// TIA Portal V16 export
// export: Created 2021-03-05T14:22:14.2551895Z, ExportSetting WithDefaults, DisplayName Totally Integrated Automation Portal, DisplayVersion V16, DisplayName TIA Portal Version Control Interface, DisplayVersion V16, DisplayName TIA Portal Openness, DisplayVersion V16, DisplayName SINAMICS Startdrive Advanced, DisplayVersion V16, DisplayName SINAMICS Startdrive G130, G150, S120, S150, SINAMICS MV, S210, DisplayVersion V16, DisplayName SINAMICS Startdrive G110M, G120, G120C, G120D, G120P, DisplayVersion V16, DisplayName STEP 7 Professional, DisplayVersion V16, DisplayName STEP 7 Safety, DisplayVersion V16, DisplayName WinCC Professional, DisplayVersion V16
TYPE "udtDigitalOutput"
// stored: IsFailsafeCompliant false
   STRUCT
      bAutoVal { ExternalVisible := 'False'; ExternalWritable := 'False'} : Bool;   // Value set by the program
      bOverrideVal { ExternalVisible := 'False'} : Bool;   // Value set by the user, tracks bAuto when bOverrideEnable=0
      bStatus { ExternalVisible := 'False'; ExternalWritable := 'False'} : Bool;   // Value being written to actual output
      bOverrideEnable { ExternalVisible := 'False'} : Bool;   // Sets bOut to bOverride
   END_STRUCT;
END_TYPE
